TYPE Symbol :
STRUCT
	info : __SYSTEM.AnyType; // varinfo?
	
	description : STRING;
END_STRUCT
END_TYPE

(* stored: Version 1.1.0.1, ProductVersion 3.1.4024.11
   DUT Symbol: Id {059f0472-13a3-4096-a372-18a255cd328a} *)
